(* Schneider Machine Expert - Basic project MINING_ORE_SORTING_COMPILE_SAFE, file version 3.0.0.0 *)
(* ProjectInformations: Name=New project *)

HARDWARE
  Cpu 0: TM221CE24R
  ModuleExtensionObject 0: TM3DI32K
  ModuleExtensionObject 1: TM3AI2H/G
  EthernetConfiguration: NetworkName=M221, IpAllocationMode=FixedAddress, IpAddress=0.0.0.0, SubnetMask=0.0.0.0
  SerialLineConfiguration: Baud=Baud19200, Parity=ParityEven, DataBits=DataBits8, StopBits=StopBits1, PhysicalMedium=PhysicalMediumRs485, TransmissionMode=TransmissionModeModbusRtu, SlaveId=1, Addressing=SlaveAddressing
  MastTask: UsePeriodScanMode=false, PeriodScan=100
  FastTask: Period=255
  CpuBehavior: StartingMode=StartAsPreviousState, AutoSaveRamOnEeprom=true, WatchdogPeriod=250

SYMBOLS  (address, symbol, comment, settings)
  %M0       AUTO_MODE  "1 automatic; 0 manual"
  %M1       START_HMI  "Remote start pulse"
  %M2       STOP_HMI  "Remote normal-stop command"
  %M3       AUTO_ENABLE  "Automatic sorting enable"
  %M10      SYSTEM_RUN  "Ore sorting run memory"
  %M11      SAFETY_OK  "Safety permissive summary"
  %M12      MANUAL_DEMAND  "Manual run demand"
  %M13      AUTO_DEMAND  "Automatic run demand"
  %M14      REJECT_BIN_FULL  "Reject-bin full interlock"
  %M20      HIGH_GRADE_LATCH  "Current parcel high grade"
  %M21      MEDIUM_GRADE_LATCH  "Current parcel medium grade"
  %M22      REJECT_LATCH  "Current parcel rejected"
  %M23      SORT_BUSY  "Sorting sequence active"
  %M24      DIVERTER_ACTIVE  "Diverter phase active"
  %M25      SEQUENCE_RESET  "Sequence-complete reset pulse"
  %M30      ALARM_ACTIVE  "Common alarm summary"
  %M40      RESET_COUNTERS  "Reset production counters"
  %S13      SB_FIRSTRUN  "Indicates the first controller cycle in RUN mode"
  %TM0      ORE_TRAVEL_TIMER  "Travel time from XRF to diverter"
  %TM1      DIVERTER_DWELL_TIMER  "Diverter actuation dwell time"
  %C0       HIGH_GRADE_TOTAL  "High-grade ore parcel total"
  %C1       MEDIUM_GRADE_TOTAL  "Medium-grade ore parcel total"
  %C2       REJECT_TOTAL  "Rejected ore parcel total"
  %I0.0     START_PB  "Local plant start pushbutton"
  %I0.1     STOP_OK  "Normal stop loop; 1 healthy"
  %I0.2     ESTOP_OK  "Safety relay feedback; 1 healthy"
  %I0.3     OL_CONVEYOR_OK  "Ore conveyor overload; 1 healthy"
  %I0.4     XRF_TRIGGER  "Ore parcel at XRF analyser"
  %I0.5     GRADE_HIGH  "High-grade classification input"
  %I0.6     GRADE_MEDIUM  "Medium-grade classification input"
  %I0.7     DIVERTER_HOME  "All diverters home and safe"
  %I0.8     SPARE_I08  "Reserved field input"
  %I0.9     SPARE_I09  "Reserved field input"
  %I0.10    SPARE_I10  "Reserved field input"
  %I0.11    SPARE_I11  "Reserved field input"
  %I0.12    SPARE_I12  "Reserved field input"
  %I0.13    SPARE_I13  "Reserved field input"
  %Q0.0     MOTOR_ORE_CONVEYOR  "Ore analyser conveyor contactor/VFD"
  %Q0.1     DIVERTER_HIGH_GRADE  "High-grade chute solenoid"
  %Q0.2     DIVERTER_MEDIUM_GRADE  "Medium-grade chute solenoid"
  %Q0.3     DIVERTER_REJECT  "Reject chute solenoid"
  %Q0.4     LAMP_RUN  "Plant running beacon"
  %Q0.5     LAMP_FAULT  "Common fault beacon"
  %Q0.6     SPARE_Q06  "Reserved output"
  %Q0.7     SPARE_Q07  "Reserved output"
  %Q0.8     SPARE_Q08  "Reserved output"
  %Q0.9     SPARE_Q09  "Reserved output"
  %I1.0     ENC_G1_GRAY_B0  "E6CP pintu 1 Gray bit 0"
  %I1.1     ENC_G1_GRAY_B1  "E6CP pintu 1 Gray bit 1"
  %I1.2     ENC_G1_GRAY_B2  "E6CP pintu 1 Gray bit 2"
  %I1.3     ENC_G1_GRAY_B3  "E6CP pintu 1 Gray bit 3"
  %I1.4     ENC_G1_GRAY_B4  "E6CP pintu 1 Gray bit 4"
  %I1.5     ENC_G1_GRAY_B5  "E6CP pintu 1 Gray bit 5"
  %I1.6     ENC_G1_GRAY_B6  "E6CP pintu 1 Gray bit 6"
  %I1.7     ENC_G1_GRAY_B7  "E6CP pintu 1 Gray bit 7"
  %I1.8     ENC_G2_GRAY_B0  "E6CP pintu 2 Gray bit 0"
  %I1.9     ENC_G2_GRAY_B1  "E6CP pintu 2 Gray bit 1"
  %I1.10    ENC_G2_GRAY_B2  "E6CP pintu 2 Gray bit 2"
  %I1.11    ENC_G2_GRAY_B3  "E6CP pintu 2 Gray bit 3"
  %I1.12    ENC_G2_GRAY_B4  "E6CP pintu 2 Gray bit 4"
  %I1.13    ENC_G2_GRAY_B5  "E6CP pintu 2 Gray bit 5"
  %I1.14    ENC_G2_GRAY_B6  "E6CP pintu 2 Gray bit 6"
  %I1.15    ENC_G2_GRAY_B7  "E6CP pintu 2 Gray bit 7"
  %I1.16    ENC_G3_GRAY_B0  "E6CP pintu 3 Gray bit 0"
  %I1.17    ENC_G3_GRAY_B1  "E6CP pintu 3 Gray bit 1"
  %I1.18    ENC_G3_GRAY_B2  "E6CP pintu 3 Gray bit 2"
  %I1.19    ENC_G3_GRAY_B3  "E6CP pintu 3 Gray bit 3"
  %I1.20    ENC_G3_GRAY_B4  "E6CP pintu 3 Gray bit 4"
  %I1.21    ENC_G3_GRAY_B5  "E6CP pintu 3 Gray bit 5"
  %I1.22    ENC_G3_GRAY_B6  "E6CP pintu 3 Gray bit 6"
  %I1.23    ENC_G3_GRAY_B7  "E6CP pintu 3 Gray bit 7"
  %I1.24    MODE_AUTO  "Selector 1=AUTO 0=MANUAL"
  %I1.25    MAN_OPEN_G1  "PB manual buka pintu 1"
  %I1.26    MAN_CLOSE_G1  "PB manual tutup pintu 1"
  %I1.27    MAN_OPEN_G2  "PB manual buka pintu 2"
  %I1.28    MAN_CLOSE_G2  "PB manual tutup pintu 2"
  %I1.29    MAN_OPEN_G3  "PB manual buka pintu 3"
  %I1.30    MAN_CLOSE_G3  "PB manual tutup pintu 3"
  %I1.31    RESET_FAULT  "PB reset fault"
  %IW2.0    LEVEL_RAW  "Sensor level 4-20 mA raw 4000-20000"  [Type=Type_4_20mA, Scope=Scope_Customized, Minimum=4000, Maximum=20000]

POU ORE_SORTING_28R_IL
  (* SectionNumber=0 *)

// Rung 0: N00_PRODUCTION_COUNTER_PRESETS
// First scan: initialize high, medium, and reject production counter presets.
  LD %S13                 (* SB_FIRSTRUN *)
  [ %C0.P := 9999 ]       (* HIGH_GRADE_TOTAL *)
  [ %C1.P := 9999 ]       (* MEDIUM_GRADE_TOTAL *)
  [ %C2.P := 9999 ]       (* REJECT_TOTAL *)
  // as ST:
  //   IF SB_FIRSTRUN THEN HIGH_GRADE_TOTAL.P := 9999; END_IF;
  //   IF SB_FIRSTRUN THEN MEDIUM_GRADE_TOTAL.P := 9999; END_IF;
  //   IF SB_FIRSTRUN THEN REJECT_TOTAL.P := 9999; END_IF;

// Rung 1
  LD %I0.1                (* STOP_OK *)
  AND %I0.2               (* ESTOP_OK *)
  AND %I0.3               (* OL_CONVEYOR_OK *)
  AND %I0.7               (* DIVERTER_HOME *)
  ANDN %M2                (* STOP_HMI *)
  ST %M11                 (* SAFETY_OK *)
  // as ST:
  //   SAFETY_OK := STOP_OK AND ESTOP_OK AND OL_CONVEYOR_OK AND DIVERTER_HOME AND NOT STOP_HMI;

// Rung 2
  LD %I0.0                (* START_PB *)
  OR %M1                  (* START_HMI *)
  OR %M10                 (* SYSTEM_RUN *)
  ANDN %M0                (* AUTO_MODE *)
  ST %M12                 (* MANUAL_DEMAND *)
  // as ST:
  //   MANUAL_DEMAND := (START_PB OR START_HMI OR SYSTEM_RUN) AND NOT AUTO_MODE;

// Rung 3
  LD %M0                  (* AUTO_MODE *)
  AND %M3                 (* AUTO_ENABLE *)
  ST %M13                 (* AUTO_DEMAND *)
  // as ST:
  //   AUTO_DEMAND := AUTO_MODE AND AUTO_ENABLE;

// Rung 4
  LD %M12                 (* MANUAL_DEMAND *)
  OR %M13                 (* AUTO_DEMAND *)
  AND %M11                (* SAFETY_OK *)
  ST %M10                 (* SYSTEM_RUN *)
  // as ST:
  //   SYSTEM_RUN := (MANUAL_DEMAND OR AUTO_DEMAND) AND SAFETY_OK;

// Rung 5
  LDR %I0.4               (* XRF_TRIGGER *)
  AND %M10                (* SYSTEM_RUN *)
  ANDN %M23               (* SORT_BUSY *)
  AND %I0.5               (* GRADE_HIGH *)
  S %M20                  (* HIGH_GRADE_LATCH *)
  // as ST:
  //   IF RISING(XRF_TRIGGER) AND SYSTEM_RUN AND NOT SORT_BUSY AND GRADE_HIGH THEN HIGH_GRADE_LATCH := TRUE; END_IF;

// Rung 6
  LDR %I0.4               (* XRF_TRIGGER *)
  AND %M10                (* SYSTEM_RUN *)
  ANDN %M23               (* SORT_BUSY *)
  ANDN %I0.5              (* GRADE_HIGH *)
  AND %I0.6               (* GRADE_MEDIUM *)
  S %M21                  (* MEDIUM_GRADE_LATCH *)
  // as ST:
  //   IF RISING(XRF_TRIGGER) AND SYSTEM_RUN AND NOT SORT_BUSY AND NOT GRADE_HIGH AND GRADE_MEDIUM THEN MEDIUM_GRADE_LATCH := TRUE; END_IF;

// Rung 7
  LDR %I0.4               (* XRF_TRIGGER *)
  AND %M10                (* SYSTEM_RUN *)
  ANDN %M23               (* SORT_BUSY *)
  ANDN %I0.5              (* GRADE_HIGH *)
  ANDN %I0.6              (* GRADE_MEDIUM *)
  S %M22                  (* REJECT_LATCH *)
  // as ST:
  //   IF RISING(XRF_TRIGGER) AND SYSTEM_RUN AND NOT SORT_BUSY AND NOT GRADE_HIGH AND NOT GRADE_MEDIUM THEN REJECT_LATCH := TRUE; END_IF;

// Rung 8
  LDR %I0.4               (* XRF_TRIGGER *)
  AND %M10                (* SYSTEM_RUN *)
  ANDN %M23               (* SORT_BUSY *)
  S %M23                  (* SORT_BUSY *)
  // as ST:
  //   IF RISING(XRF_TRIGGER) AND SYSTEM_RUN AND NOT SORT_BUSY THEN SORT_BUSY := TRUE; END_IF;

// Rung 9
  BLK %TM0                (* ORE_TRAVEL_TIMER *)
  LD %M23                 (* SORT_BUSY *)
  ANDN %M24               (* DIVERTER_ACTIVE *)
  IN
  END_BLK
  // as ST:
  //   ORE_TRAVEL_TIMER(IN := SORT_BUSY AND NOT DIVERTER_ACTIVE);

// Rung 10
  LD %TM0.Q               (* ORE_TRAVEL_TIMER *)
  S %M24                  (* DIVERTER_ACTIVE *)
  // as ST:
  //   IF ORE_TRAVEL_TIMER.Q THEN DIVERTER_ACTIVE := TRUE; END_IF;

// Rung 11
  BLK %TM1                (* DIVERTER_DWELL_TIMER *)
  LD %M24                 (* DIVERTER_ACTIVE *)
  IN
  END_BLK
  // as ST:
  //   DIVERTER_DWELL_TIMER(IN := DIVERTER_ACTIVE);

// Rung 12
  LD %M10                 (* SYSTEM_RUN *)
  AND %M11                (* SAFETY_OK *)
  ANDN %M24               (* DIVERTER_ACTIVE *)
  ANDN %M14               (* REJECT_BIN_FULL *)
  ST %Q0.0                (* MOTOR_ORE_CONVEYOR *)
  // as ST:
  //   MOTOR_ORE_CONVEYOR := SYSTEM_RUN AND SAFETY_OK AND NOT DIVERTER_ACTIVE AND NOT REJECT_BIN_FULL;

// Rung 13
  LD %M24                 (* DIVERTER_ACTIVE *)
  AND %M20                (* HIGH_GRADE_LATCH *)
  AND %M11                (* SAFETY_OK *)
  ST %Q0.1                (* DIVERTER_HIGH_GRADE *)
  // as ST:
  //   DIVERTER_HIGH_GRADE := DIVERTER_ACTIVE AND HIGH_GRADE_LATCH AND SAFETY_OK;

// Rung 14
  LD %M24                 (* DIVERTER_ACTIVE *)
  AND %M21                (* MEDIUM_GRADE_LATCH *)
  AND %M11                (* SAFETY_OK *)
  ST %Q0.2                (* DIVERTER_MEDIUM_GRADE *)
  // as ST:
  //   DIVERTER_MEDIUM_GRADE := DIVERTER_ACTIVE AND MEDIUM_GRADE_LATCH AND SAFETY_OK;

// Rung 15
  LD %M24                 (* DIVERTER_ACTIVE *)
  AND %M22                (* REJECT_LATCH *)
  AND %M11                (* SAFETY_OK *)
  ST %Q0.3                (* DIVERTER_REJECT *)
  // as ST:
  //   DIVERTER_REJECT := DIVERTER_ACTIVE AND REJECT_LATCH AND SAFETY_OK;

// Rung 16
  BLK %C0                 (* HIGH_GRADE_TOTAL *)
  LD %M40                 (* RESET_COUNTERS *)
  R
  LD %TM1.Q               (* DIVERTER_DWELL_TIMER *)
  AND %M20                (* HIGH_GRADE_LATCH *)
  CU
  END_BLK
  // as ST:
  //   HIGH_GRADE_TOTAL(R := RESET_COUNTERS, CU := DIVERTER_DWELL_TIMER.Q AND HIGH_GRADE_LATCH);

// Rung 17
  BLK %C1                 (* MEDIUM_GRADE_TOTAL *)
  LD %M40                 (* RESET_COUNTERS *)
  R
  LD %TM1.Q               (* DIVERTER_DWELL_TIMER *)
  AND %M21                (* MEDIUM_GRADE_LATCH *)
  CU
  END_BLK
  // as ST:
  //   MEDIUM_GRADE_TOTAL(R := RESET_COUNTERS, CU := DIVERTER_DWELL_TIMER.Q AND MEDIUM_GRADE_LATCH);

// Rung 18
  BLK %C2                 (* REJECT_TOTAL *)
  LD %M40                 (* RESET_COUNTERS *)
  R
  LD %TM1.Q               (* DIVERTER_DWELL_TIMER *)
  AND %M22                (* REJECT_LATCH *)
  CU
  END_BLK
  // as ST:
  //   REJECT_TOTAL(R := RESET_COUNTERS, CU := DIVERTER_DWELL_TIMER.Q AND REJECT_LATCH);

// Rung 19
  LD %TM1.Q               (* DIVERTER_DWELL_TIMER *)
  ST %M25                 (* SEQUENCE_RESET *)
  // as ST:
  //   SEQUENCE_RESET := DIVERTER_DWELL_TIMER.Q;

// Rung 20
  LD %M25                 (* SEQUENCE_RESET *)
  R %M24                  (* DIVERTER_ACTIVE *)
  // as ST:
  //   IF SEQUENCE_RESET THEN DIVERTER_ACTIVE := FALSE; END_IF;

// Rung 21
  LD %M25                 (* SEQUENCE_RESET *)
  R %M23                  (* SORT_BUSY *)
  // as ST:
  //   IF SEQUENCE_RESET THEN SORT_BUSY := FALSE; END_IF;

// Rung 22
  LD %M25                 (* SEQUENCE_RESET *)
  R %M20                  (* HIGH_GRADE_LATCH *)
  // as ST:
  //   IF SEQUENCE_RESET THEN HIGH_GRADE_LATCH := FALSE; END_IF;

// Rung 23
  LD %M25                 (* SEQUENCE_RESET *)
  R %M21                  (* MEDIUM_GRADE_LATCH *)
  // as ST:
  //   IF SEQUENCE_RESET THEN MEDIUM_GRADE_LATCH := FALSE; END_IF;

// Rung 24
  LD %M25                 (* SEQUENCE_RESET *)
  R %M22                  (* REJECT_LATCH *)
  // as ST:
  //   IF SEQUENCE_RESET THEN REJECT_LATCH := FALSE; END_IF;

// Rung 25
  LDN %M11                (* SAFETY_OK *)
  OR %M14                 (* REJECT_BIN_FULL *)
  ST %M30                 (* ALARM_ACTIVE *)
  // as ST:
  //   ALARM_ACTIVE := NOT SAFETY_OK OR REJECT_BIN_FULL;

// Rung 26
  LD %M10                 (* SYSTEM_RUN *)
  ANDN %M30               (* ALARM_ACTIVE *)
  ST %Q0.4                (* LAMP_RUN *)
  // as ST:
  //   LAMP_RUN := SYSTEM_RUN AND NOT ALARM_ACTIVE;

// Rung 27
  LD %M30                 (* ALARM_ACTIVE *)
  ST %Q0.5                (* LAMP_FAULT *)
  // as ST:
  //   LAMP_FAULT := ALARM_ACTIVE;
